FUNCTION_BLOCK ThreeConveyorInput (* Composite Function Block Type *)
  (* Standard: 61499-2 *)
  (* Version 0.2, 2003-12-05, JHC, Rockwell Automation, Renamed from NEWCOMPFB. *)
  (* Version 0.1, 2002-01-08, JHC, Rockwell Automation, Added DLY FB as example. *)
  (* Version 0.0, 2000-05-27, JHC, Rockwell Automation *)
  (* Compiler header: package fb.rt.cs725;import fb.rt.vhmi.*; *)
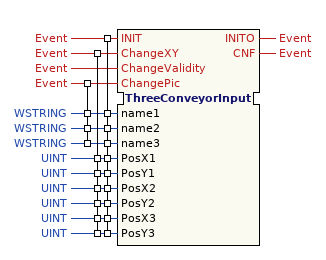
  EVENT_INPUT
    INIT WITH name1, name2, name3, PosX1, PosY1, PosX2, PosY2, PosX3, PosY3; (* Initialization Request *)
    ChangeXY WITH PosX1, PosY1, PosX2, PosY2, PosX3, PosY3; (* Normal Execution Request *)
    ChangeValidity;
    ChangePic WITH name1, name2, name3;
  END_EVENT
  EVENT_OUTPUT
    INITO; (* Initialization Confirm *)
    CNF; (* Execution Confirmation *)
  END_EVENT
  VAR_INPUT
    name1 : WSTRING;
    name2 : WSTRING;
    name3 : WSTRING;
    PosX1 : UINT;
    PosY1 : UINT;
    PosX2 : UINT;
    PosY2 : UINT;
    PosX3 : UINT;
    PosY3 : UINT;
  END_VAR
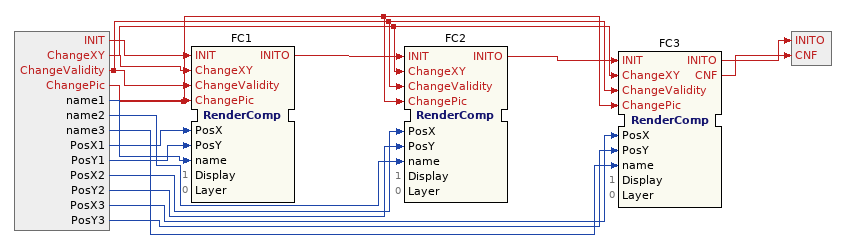
  FBS
    FC1 : RenderComp(Display := 1, Layer := 0);
    FC2 : RenderComp(Display := 1, Layer := 0);
    FC3 : RenderComp(Display := 1, Layer := 0);
  END_FBS
  EVENT_CONNECTIONS
    INIT TO FC1.INIT;
    ChangeXY TO FC1.ChangeXY;
    ChangeValidity TO FC1.ChangeValidity;
    ChangePic TO FC1.ChangePic;
    FC1.INITO TO FC2.INIT;
    FC2.INITO TO FC3.INIT;
    FC3.INITO TO INITO;
    FC3.CNF TO CNF;
    ChangeXY TO FC2.ChangeXY;
    ChangeValidity TO FC2.ChangeValidity;
    ChangePic TO FC2.ChangePic;
    ChangeXY TO FC3.ChangeXY;
    ChangeValidity TO FC3.ChangeValidity;
    ChangePic TO FC3.ChangePic;
  END_CONNECTIONS
  DATA_CONNECTIONS
    PosX1 TO FC1.PosX;
    PosY1 TO FC1.PosY;
    PosX2 TO FC2.PosX;
    PosY2 TO FC2.PosY;
    PosX3 TO FC3.PosX;
    PosY3 TO FC3.PosY;
    name1 TO FC1.name;
    name2 TO FC2.name;
    name3 TO FC3.name;
  END_CONNECTIONS
END_FUNCTION_BLOCK
